(* IEC 61131-3 sources: PraktykiBr/BottlePlant2/Software/Code/RecipeControl/RecipeCtrl, 2 files *)

(* ---- Main.st ---- *)
PROGRAM _INIT
	(* Insert code here *)
	Recipe.RecipeXml.Enable:=TRUE;
	Recipe.RecipeUI.Enable:=TRUE;
	Recipe.RecipeRegPar.Enable:=TRUE;
	Recipe.FileManagerUI.Enable:=TRUE;

	Recipe.State:=STATE_WAIT_RECIPE;
END_PROGRAM

PROGRAM _CYCLIC
	(* Insert code here *)
	Recipe.RecipeXml.MpLink:=ADR(gRecipeXml);
	Recipe.RecipeXml.DeviceName:=ADR(Recipe.RecipeData.DeviceName);
	Recipe.RecipeXml.FileName:=ADR('recipe');

	Recipe.RecipeUI.MpLink:=ADR(gRecipeXml);
	Recipe.RecipeUI.UIConnect:=ADR(Recipe.RecipeUIConnect);

	Recipe.RecipeUISetup.Confirmation.RecipeLoad:=TRUE;
	Recipe.RecipeUISetup.Confirmation.RecipeDelete:=TRUE;
	Recipe.RecipeUISetup.Confirmation.RecipeSave:=TRUE;
	Recipe.RecipeUISetup.Confirmation.RecipeCreate:=TRUE;
	Recipe.RecipeUISetup.Confirmation.RecipeRename:=TRUE;
	Recipe.RecipeUI.UISetup:=Recipe.RecipeUISetup;

	Recipe.RecipeRegPar.MpLink:=ADR(gRecipeXml);
	Recipe.RecipeRegPar.PVName:=ADR('gRecipeValues');

	Recipe.FileManagerUI.MpLink:=ADR(gFileManagerUI);
	Recipe.FileManagerUI.UIConnect:=ADR(Recipe.FileManagerUIConnect);
	Recipe.FileManagerUI.UISetup:=Recipe.FileManagerSetup;

	Recipe.FileManagerUIConnect.DeviceList.DeviceNames[0]:=Recipe.RecipeData.DeviceName;

	(* Maszyna stanów kontrolująca zapisywanie i wczytywanie z recipe do struktury  *)
	CASE Recipe.State OF
		STATE_WAIT_RECIPE:
			(* Jesli receptura jest wczytywana, przejdz do odpowiedniego stanu  *)
			IF Recipe.RecipeUIConnect.Status=mpRECIPE_UI_STATUS_LOAD THEN
				Recipe.State:=STATE_LOAD_RECIPE;
			(* Jeśli wyskoczył message box proszący o potwierdzenie zapisu struktury do recipe, przejdz do odpowiedniego stanu  *)
			ELSIF Recipe.RecipeUIConnect.MessageBox.Type=mpRECIPE_UI_MSG_CONFIRM_SAVE THEN
				Recipe.State:=STATE_SAVE_RECIPE;
			END_IF;
		STATE_LOAD_RECIPE:
			(* Jesli bloczek oczekuje na cmd tzn że zostało wczytanie do struktury i można zaimplementować zmiany ze struktury do camseq *)
			IF Recipe.RecipeUIConnect.Status=mpRECIPE_UI_STATUS_IDLE THEN
				gRecipeLoaded:=TRUE; //flaga informująca że jakakolwiek receptura została waczytana

				(* Aktualizacja zmiennych z GUI *)
				uiRecipeBottlePerMinute := gRecipeValues[1].Velocity;
				uiRecipeBottlePerHour := gRecipeValues[1].Velocity;
				uiBottlePerHour:=gRecipeValues[1].Velocity;
				uiBottlePerMinute:=gRecipeValues[1].Velocity;

				(* Aktualizacja parametrów sequencera *)
				gAxes.Ctrl.MpTransporterAxisPar.Velocity:=gRecipeValues[1].Velocity;
				gCamSequencer.Ctrl.MpAxisCamSequencerPar_1.Configuration.State[1].CamProfileIndex:=gRecipeValues[1].CamProfileIndex;
				gCamSequencer.Ctrl.MpAxisCamSequencerPar_1.Configuration.State[1].MasterCompDistance:=gRecipeValues[1].MasterCompDistance;
				gCamSequencer.Ctrl.MpAxisCamSequencerPar_1.Configuration.State[1].SlaveCompDistance:=gRecipeValues[1].SlaveComDistance;
				gCamSequencer.Ctrl.MpAxisCamSequencerPar_1.Configuration.State[1].MasterFactor:=gRecipeValues[1].MasterFactor;
				gCamSequencer.Ctrl.MpAxisCamSequencerPar_1.Configuration.State[1].SlaveFactor:=gRecipeValues[1].SlaveFactor;

				gCamSequencer.Ctrl.MpAxisCamSequencerPar_1.Configuration.State[2].CamProfileIndex:=gRecipeValues[2].CamProfileIndex;
				gCamSequencer.Ctrl.MpAxisCamSequencerPar_1.Configuration.State[2].MasterCompDistance:=gRecipeValues[2].MasterCompDistance;
				gCamSequencer.Ctrl.MpAxisCamSequencerPar_1.Configuration.State[2].SlaveCompDistance:=gRecipeValues[2].SlaveComDistance;
				gCamSequencer.Ctrl.MpAxisCamSequencerPar_1.Configuration.State[2].MasterFactor:=gRecipeValues[2].MasterFactor;
				gCamSequencer.Ctrl.MpAxisCamSequencerPar_1.Configuration.State[2].SlaveFactor:=gRecipeValues[2].SlaveFactor;

				(* Update dokonanych zmian -> Update musi dokonać się w odpowiednim state aby nie popsuć pracy  *)
				IF gCamSequencer.Ctrl.MpAxisCamSequencer_0.StartSequence=TRUE AND gCamSequencer.Ctrl.MpAxisCamSequencer_0.ActualStateIndex=2 THEN
					gCamSequencer.Ctrl.MpAxisCamSequencer_1.Update:=TRUE;
					gAxes.Cmd.Auto.Update:=TRUE;
					Recipe.State:=STATE_WAIT_RECIPE;
				ELSIF gCamSequencer.Ctrl.MpAxisCamSequencer_0.StartSequence=FALSE THEN
					gCamSequencer.Ctrl.MpAxisCamSequencer_1.Update:=TRUE;
					gAxes.Cmd.Auto.Update:=TRUE;
					Recipe.State:=STATE_WAIT_RECIPE;
				END_IF
			END_IF;

		STATE_SAVE_RECIPE:
			(* Zapisanie aktualnych parametrów sequencera do struktury -> aktualizacja tylko wtedy gdy wyskoczy message box *)
				gRecipeValues[1].Velocity:=gAxes.Ctrl.MpTransporterAxisPar.Velocity;
				gRecipeValues[1].CamProfileIndex:=gCamSequencer.Ctrl.MpAxisCamSequencerPar_1.Configuration.State[1].CamProfileIndex;
				gRecipeValues[1].MasterCompDistance:=gCamSequencer.Ctrl.MpAxisCamSequencerPar_1.Configuration.State[1].MasterCompDistance;
				gRecipeValues[1].SlaveComDistance:=gCamSequencer.Ctrl.MpAxisCamSequencerPar_1.Configuration.State[1].SlaveCompDistance;
				gRecipeValues[1].MasterFactor:=gCamSequencer.Ctrl.MpAxisCamSequencerPar_1.Configuration.State[1].MasterFactor;
				gRecipeValues[1].SlaveFactor:=gCamSequencer.Ctrl.MpAxisCamSequencerPar_1.Configuration.State[1].SlaveFactor;

				gRecipeValues[2].Velocity:=gAxes.Ctrl.MpTransporterAxisPar.Velocity;
				gRecipeValues[2].CamProfileIndex:=gCamSequencer.Ctrl.MpAxisCamSequencerPar_1.Configuration.State[2].CamProfileIndex;
				gRecipeValues[2].MasterCompDistance:=gCamSequencer.Ctrl.MpAxisCamSequencerPar_1.Configuration.State[2].MasterCompDistance;
				gRecipeValues[2].SlaveComDistance:=gCamSequencer.Ctrl.MpAxisCamSequencerPar_1.Configuration.State[2].SlaveCompDistance;
				gRecipeValues[2].MasterFactor:=gCamSequencer.Ctrl.MpAxisCamSequencerPar_1.Configuration.State[2].MasterFactor;
				gRecipeValues[2].SlaveFactor:=gCamSequencer.Ctrl.MpAxisCamSequencerPar_1.Configuration.State[2].SlaveFactor;
				Recipe.State:=STATE_WAIT_RECIPE;

	END_CASE;

	Recipe.RecipeXml();
	Recipe.RecipeRegPar();
	Recipe.RecipeUI();
	Recipe.FileManagerUI();
END_PROGRAM

PROGRAM _EXIT
	(* Insert code here *)

END_PROGRAM

(* ---- Variables.var ---- *)
VAR
	Recipe : RecipeCtrlType;
END_VAR

VAR CONSTANT

END_VAR
